// SIMATIC S7-200 project (STEP 7-Micro/WIN), CPU 221 REL 01.10

ORGANIZATION_BLOCK 主程序:OB1
TITLE=程序注释
BEGIN
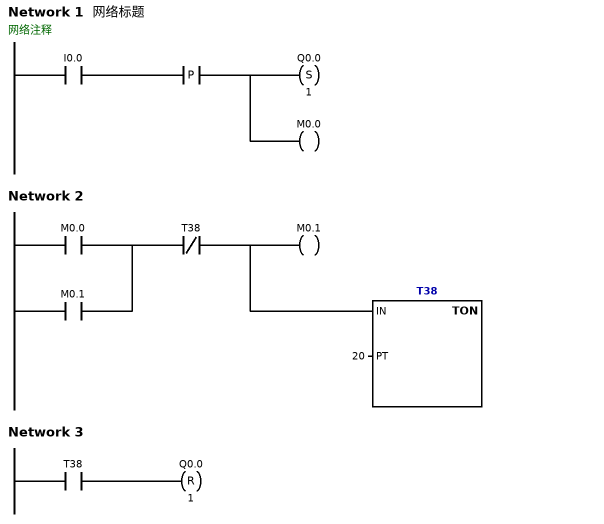
Network 1 // 网络标题
// 网络注释
LD     I0.0
EU
S      Q0.0, 1
=      M0.0
Network 2
LD     M0.0
O      M0.1
AN     T38
=      M0.1
TON    T38, 20
Network 3
LD     T38
R      Q0.0, 1
END_ORGANIZATION_BLOCK
